{attribute 'qualified_only'}
{attribute 'to_string'}
TYPE E_HVAL_STATUS :
(
	NONE := 0,
	GREEN_HV_OFF := 1,
	BLINKING_RED_HV_ON := 2
) USINT;
END_TYPE

(* stored: Version 1.1.0.1
   DUT E_HVAL_STATUS: Id {56ddce06-d350-46b7-bb38-76016c413049} *)
